FUNCTION_BLOCK ComparisonFunctionsTest EXTENDS TcUnit.FB_TestSuite
VAR
END_VAR

DataEqualsFunction();

METHOD DataEqualsFunction : BOOL
VAR
	data1 : INT;
	data2 : INT;
END_VAR
TcUnit.TEST('Data equals');

data1 := 42;
data2 := 0;

AssertEquals_BOOL(
	Expected := FALSE,
	Actual := DataEquals(data1, data2),
	Message := 'Data should not be equal');

data2 := data1;

AssertEquals_BOOL(
	Expected := TRUE,
	Actual := DataEquals(data1, data2),
	Message := 'Data should be equal');

TEST_FINISHED();
END_METHOD

END_FUNCTION_BLOCK

(* stored: Version 1.1.0.1, ProductVersion 3.1.4024.15
   POU ComparisonFunctionsTest: Id {c66b0d62-1fe5-0058-3582-deef21484393}, SpecialFunc None
   Method DataEqualsFunction: Id {69d32c70-5f4c-079b-1fcc-553ae9f1ddce} *)
